ADAPTER BOOL_Event (* Adapter Interface *)
  (* Standard: 61499-1 *)
  (* Version 0.0, 12/12/2023, Cheyan, Schneider Electric *)
  PACKAGE Main;
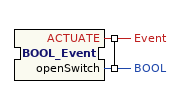
  EVENT_OUTPUT
    ACTUATE WITH openSwitch; (* Confirmation from Plug *)
  END_EVENT
  VAR_OUTPUT
    openSwitch : BOOL; (* Confirmation Data from Plug *)
  END_VAR
  SERVICE SOCKET/PLUG
    SEQUENCE request_confirm
      SOCKET.REQ(REQD) -> PLUG.REQ(REQD);
      PLUG.ACTUATE(openSwitch) -> SOCKET.ACTUATE(openSwitch);
    END_SEQUENCE
    SEQUENCE indication_response
      PLUG.IND(INDD) -> SOCKET.IND(INDD);
      SOCKET.RSP(RSPD) -> PLUG.RSP(RSPD);
    END_SEQUENCE
  END_SERVICE
END_ADAPTER
